// Mitsubishi GX Works2 project: BookEX6_13 Timer   PLC: Q13UDV

// global labels: Global
VAR_GLOBAL
  bVar0 AT M5000 : BOOL;
  abArray0 AT M5010 : ARRAY [0..49] OF BOOL;
  sStr0 AT D5000 : STRING[199];
  sStr1 AT D5100 : STRING[199];
  sStr2 AT D5200 : STRING[199];
  sStr3 AT D5300 : STRING[199];
  sStr4 AT D5400 : STRING[199];
  sStr5 AT D5500 : STRING[199];
  sStr6 AT D5600 : STRING[199];
  sStr7 AT D5700 : STRING[199];
  sStr8 AT D5800 : STRING[199];
  sStr9 AT D5900 : STRING[199];
  iVar0 AT D4500 : INT;
  iVar1 AT D4501 : INT;
  iVar2 AT D4502 : INT;
  iVar3 AT D4503 : INT;
  iVar4 AT D4504 : INT;
  iVar5 AT D4505 : INT;
  iVar6 AT D4506 : INT;
  iVar7 AT D4507 : INT;
  iVar8 AT D4508 : INT;
  iVar9 AT D4509 : INT;
  dVar0 AT D4510 : DINT;
  dVar1 AT D4512 : DINT;
  dVar2 AT D4514 : DINT;
  dVar3 AT D4516 : DINT;
  dVar4 AT D4518 : DINT;
  dVar5 AT D4520 : DINT;
  dVar6 AT D4522 : DINT;
  dVar7 AT D4524 : DINT;
  dVar8 AT D4526 : DINT;
  dVar9 AT D4528 : DINT;
  wVar0 AT D4530 : WORD;
  wVar1 AT D4531 : WORD;
  wVar2 AT D4532 : WORD;
  wVar3 AT D4533 : WORD;
  wVar4 AT D4534 : WORD;
  wVar5 AT D4535 : WORD;
  wVar6 AT D4536 : WORD;
  wVar7 AT D4537 : WORD;
  wVar8 AT D4538 : WORD;
  wVar9 AT D4539 : WORD;
  dwVar0 AT D4540 : DWORD;
  dwVar1 AT D4542 : DWORD;
  dwVar2 AT D4544 : DWORD;
  dwVar3 AT D4546 : DWORD;
  dwVar4 AT D4548 : DWORD;
  dwVar5 AT D4550 : DWORD;
  dwVar6 AT D4552 : DWORD;
  dwVar7 AT D4554 : DWORD;
  dwVar8 AT D4556 : DWORD;
  dwVar9 AT D4558 : DWORD;
  fsVar0 AT D4560 : REAL;
  fsVar1 AT D4562 : REAL;
  fsVar2 AT D4564 : REAL;
  fsVar3 AT D4566 : REAL;
  fsVar4 AT D4568 : REAL;
  fsVar5 AT D4570 : REAL;
  fsVar6 AT D4572 : REAL;
  fsVar7 AT D4574 : REAL;
  fsVar8 AT D4576 : REAL;
  fsVar9 AT D4578 : REAL;
  fdVar0 AT D4580 : LREAL;
  tTime0 AT D4620 : TIME;
  tTime1 AT D4622 : TIME;
  tTime2 AT D4624 : TIME;
  tTime3 AT D4626 : TIME;
  tTime4 AT D4628 : TIME;
  tTime5 AT D4630 : TIME;
  tTime6 AT D4632 : TIME;
  tTime7 AT D4634 : TIME;
  tTime8 AT D4636 : TIME;
  tTime9 AT D4638 : TIME;
  tTime10 AT D4640 : TIME;
  bVar1 AT M5001 : BOOL;
  bVar2 AT M5002 : BOOL;
  bVar3 AT M5003 : BOOL;
  bVar4 AT M5004 : BOOL;
  bVar5 AT M5005 : BOOL;
  bVar6 AT M5006 : BOOL;
  bVar7 AT M5007 : BOOL;
  bVar8 AT M5008 : BOOL;
  bVar9 AT M5009 : BOOL;
  abArray1 AT M5060 : ARRAY [0..49] OF BOOL;
  abArray2 AT M5110 : ARRAY [0..49] OF BOOL;
  abArray3 AT M5160 : ARRAY [0..49] OF BOOL;
  abArray4 AT M5210 : ARRAY [0..49] OF BOOL;
  abArray5 AT M5260 : ARRAY [0..49] OF BOOL;
  abArray6 AT M5310 : ARRAY [0..49] OF BOOL;
  abArray7 AT M5360 : ARRAY [0..49] OF BOOL;
  abArray8 AT M5410 : ARRAY [0..49] OF BOOL;
  abArray9 AT M5460 : ARRAY [0..49] OF BOOL;
  fdVar1 AT D4584 : LREAL;
  fdVar2 AT D4588 : LREAL;
  fdVar3 AT D4592 : LREAL;
  fdVar4 AT D4596 : LREAL;
  fdVar5 AT D4600 : LREAL;
  fdVar6 AT D4604 : LREAL;
  fdVar7 AT D4608 : LREAL;
  fdVar8 AT D4612 : LREAL;
  fdVar9 AT D4616 : LREAL;
  aSendData1 AT D100 : ARRAY [0..9] OF INT;
  aiTxData AT D4000 : ARRAY [0..99] OF INT;
  aiRxData AT D4100 : ARRAY [0..99] OF INT;
  iOpenOK AT D3900 : INT;
  iOpenERR AT D3901 : INT;
  iSendOK AT D3902 : INT;
  iSendERR AT D3903 : INT;
  iCloseOK AT D3906 : INT;
  iCloseERR AT D3907 : INT;
  iRecvOK AT D3904 : INT;
  iRecvERR AT D3905 : INT;
  aiTxData2 AT D4200 : ARRAY [0..99] OF INT;
  aiRxData2 AT D4300 : ARRAY [0..99] OF INT;
  iOpenOK2 AT D3908 : INT;
  iOpenERR2 AT D3909 : INT;
  iSendOK2 AT D3910 : INT;
  iSendERR2 AT D3911 : INT;
  iRecvOK2 AT D3912 : INT;
  iRecvERR2 AT D3913 : INT;
  iCloseOK2 AT D3914 : INT;
  iCloseERR2 AT D3915 : INT;
  iEOpenComp AT D3916 : INT;
  iEOpenReq AT D3917 : INT;
  iERecvFlag AT D3918 : INT;
  iOpenCode AT D3919 : INT;
  iSendCode AT D3920 : INT;
  iRecvCode AT D3921 : INT;
  iCloseCode AT D3922 : INT;
  iOpenCode2 AT D3923 : INT;
  iSendCode2 AT D3924 : INT;
  iRecvCode2 AT D3925 : INT;
  iCloseCode2 AT D3926 : INT;
  aRecvData1 AT D110 : ARRAY [0..9] OF INT;
  aSendData2 AT D120 : ARRAY [0..9] OF INT;
  aRecvData2 AT D130 : ARRAY [0..9] OF INT;
END_VAR
// user libraries (not included): HMI

FUNCTION_BLOCK BlinkFlag
VAR_INPUT
  b_EN : BOOL;
END_VAR
VAR_OUTPUT
  b_ENO : BOOL;
END_VAR
VAR
  bBlink : BOOL;
  fbTimer1 : TON;
  fbTimer2 : TON;
  BlinkTime : TIME;
END_VAR
VAR_OUTPUT
  t_ON : TIME;
  t_OFF : TIME;
END_VAR
VAR_INPUT
  i_Duty : INT;
END_VAR
VAR_OUTPUT
  b_Q : BOOL;
END_VAR
b_ENO := b_EN;
IF NOT b_EN THEN
	b_Q := FALSE;
	bBlink := FALSE;
	fbTimer1(IN:=FALSE);
	fbTimer2(IN:=FALSE);
	RETURN;
END_IF;
BlinkTime := INT_TO_TIME(i_Duty*100/2);
IF bBlink THEN
		fbTimer1(IN := TRUE , PT:=BlinkTime);
		IF fbTimer1.Q THEN
			bBlink := FALSE;
			fbTimer1(IN:=FALSE);
		END_IF;
ELSE
		fbTimer2(IN := TRUE , PT:=BlinkTime);
		IF fbTimer2.Q THEN
			bBlink := TRUE;
			fbTimer2(IN:=FALSE);
		END_IF;
END_IF;
b_Q := bBlink;
t_ON := fbTimer2.ET;
t_OFF := fbTimer1.ET;
END_FUNCTION_BLOCK

FUNCTION_BLOCK CntClick
VAR_INPUT
  b_IN : BOOL;
  i_IN : INT;
  t_Time : TIME;
END_VAR
VAR_OUTPUT
  b_Q : BOOL;
END_VAR
VAR
  oldIN : BOOL;
  iCnt : INT;
  fbTP : TP;
END_VAR
VAR_OUTPUT
  t_ET : TIME;
  i_Cnt : INT;
END_VAR
;
b_Q := FALSE;

IF b_IN AND NOT oldIN AND NOT fbTP.Q THEN
	iCnt := 1;
ELSIF fbTP.Q AND b_IN AND NOT oldIN THEN
	iCnt := iCnt + 1;
ELSIF NOT fbTP.Q THEN
	b_Q := iCnt = i_IN;
	iCnt := 0;
END_IF;

oldIN := b_IN;
fbTP(IN := b_IN, PT := t_Time);
t_ET := fbTP.ET;
i_Cnt := iCnt;
END_FUNCTION_BLOCK

FUNCTION_BLOCK DelayOut
VAR_INPUT
  b_SET : BOOL;
  b_RST : BOOL;
  b_IN : BOOL;
  t_Time : TIME;
END_VAR
VAR_OUTPUT
  b_Q : BOOL;
END_VAR
VAR
  fbTON : TON;
  bOld : BOOL;
END_VAR
;
IF fbTON.Q THEN b_Q := FALSE; END_IF;
IF b_RST THEN
	b_Q := FALSE;
ELSIF b_SET THEN
	b_Q := TRUE;
ELSIF b_IN AND NOT bOld THEN
	b_Q := TRUE; 
END_IF;
bOld := b_IN;
IF t_Time > T#0s THEN fbTON(IN := b_Q, PT := t_Time); END_IF;
END_FUNCTION_BLOCK

FUNCTION_BLOCK FlashLamp
VAR_INPUT
  t_OnTime : TIME;
  t_OffTime : TIME;
END_VAR
VAR_OUTPUT
  b_Lamp : BOOL;
END_VAR
VAR
  bFeed : BOOL;
  TON_1 : TON;
  TON_2 : TON;
END_VAR
VAR_OUTPUT
  t_Time0 : TIME;
  t_Time1 : TIME;
END_VAR
(* structured ladder/FBD written out as ST: instructions are called as NAME(EN, inputs, outputs); _pN, _eN, _tN stand for wires *)
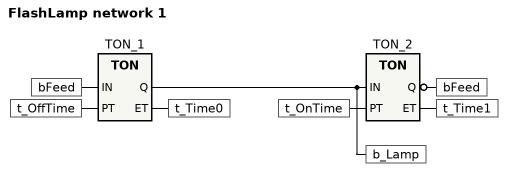
(* network 1 *)
TON_1(IN := bFeed, PT := t_OffTime, ET => t_Time0);
b_Lamp := TON_1.Q;
TON_2(IN := TON_1.Q, PT := t_OnTime, ET => t_Time1);
bFeed := NOT TON_2.Q;
END_FUNCTION_BLOCK

FUNCTION_BLOCK Flicker
VAR_INPUT
  t_Duty : TIME;
END_VAR
VAR_OUTPUT
  b_Lamp1 : BOOL;
  b_Lamp2 : BOOL;
END_VAR
VAR
  bRes : BOOL;
  iInterval : INT;
  tTimer0 : TIMER;
  tTimer1 : TIMER;
END_VAR
;
iInterval := TIME_TO_INT(t_Duty) / 100;
bResult := OUT_T(NOT tTimer1.S, tTimer0, iInterval);
bResult := OUT_T(tTimer0.S, tTimer1, iInterval);
b_Lamp1 := tTimer0.S;
b_Lamp2 :=   NOT tTimer0.S;
END_FUNCTION_BLOCK

FUNCTION_BLOCK HeartBeat
VAR_INPUT
  t_TxTime : TIME;
END_VAR
VAR_OUTPUT
  b_ENO : BOOL;
  b_TxFlag : BOOL;
END_VAR
VAR
  SeqTx : INT;
  fbTxTimer : TON;
END_VAR
VAR_INPUT
  t_RxTime : TIME;
  b_RxFlag : BOOL;
END_VAR
VAR_OUTPUT
  b_RxError : BOOL;
END_VAR
VAR
  fbRxTimer : TON;
  oldRxFlag : BOOL;
END_VAR
VAR_INPUT
  b_EN : BOOL;
END_VAR
VAR_OUTPUT
  b_TxChanged : BOOL;
END_VAR
;
b_ENO := b_EN;
IF NOT b_EN THEN
	SeqTx := 0;
	b_TxFlag := FALSE;
	b_RxError := FALSE;
	RETURN;
END_IF;
	
CASE SeqTx OF
			0 : 
				b_TxFlag := TRUE;
				SeqTx := 1;
				b_TxChanged := TRUE;
			1 : 
				b_TxChanged := FALSE;
				fbTxTimer(IN := TRUE , PT := t_TxTime);
				IF fbTxTimer.Q THEN
					fbTxTimer(IN := FALSE);
					SeqTx := 2;
				END_IF;
			2 : 
				b_TxFlag := FALSE;
				SeqTx := 3;
				b_TxChanged := TRUE;
			3 : 
				b_TxChanged := FALSE;
				fbTxTimer(IN := TRUE , PT := t_TxTime);
				IF fbTxTimer.Q THEN
					fbTxTimer(IN := FALSE);
					SeqTx := 0;
				END_IF;
ELSE
			    SeqTx := 0;
END_CASE;

IF b_RxFlag = oldRxFlag THEN
			fbRxTimer(IN := TRUE ,  PT := t_RxTime);
			IF fbRxTimer.Q THEN
				fbRxTimer(IN := FALSE);
				b_RxError := TRUE;
			END_IF;
ELSE
			fbRxTimer(IN := FALSE);
			oldRxFlag := b_RxFlag;
			b_RxError := FALSE;
END_IF;
END_FUNCTION_BLOCK

FUNCTION_BLOCK Interlock
VAR_INPUT
  b_IN1 : BOOL;
  b_IN2 : BOOL;
  t_Time : TIME;
END_VAR
VAR_OUTPUT
  b_Q1 : BOOL;
  b_Q2 : BOOL;
END_VAR
VAR
  fbTOF1 : TOF;
  fbTOF2 : TOF;
END_VAR
VAR_OUTPUT
  t_ET1 : TIME;
  t_ET2 : TIME;
END_VAR
;
fbTOF1(IN := b_IN1, PT := t_Time);
fbTOF2(IN := b_IN2, PT := t_Time);

b_Q1 := b_IN1 AND NOT fbTOF2.Q;
b_Q2 := b_IN2 AND NOT fbTOF1.Q;
t_ET1 := fbTOF1.ET;
t_ET2 := fbTOF2.ET;
END_FUNCTION_BLOCK

FUNCTION_BLOCK TONOF
VAR_INPUT
  b_IN : BOOL;
  t_ON : TIME;
  t_OFF : TIME;
END_VAR
VAR_OUTPUT
  b_Q : BOOL;
END_VAR
VAR
  fbTON : TON;
  bOld : BOOL;
  bMode : BOOL;
END_VAR
VAR_OUTPUT
  t_ET : TIME;
END_VAR
;
IF b_IN XOR bOld THEN
  fbTON(IN := FALSE, PT := SEL(b_IN, t_OFF, t_ON));
  bMode := b_IN;
  bOld := b_IN;
END_IF;
fbTON(IN := TRUE);
IF fbTON.Q THEN 
	b_Q := bMode;
END_IF;
t_ET := fbTON.ET;
END_FUNCTION_BLOCK

PROGRAM ExBlink
VAR
  HMI03_1 : HMI03;
  BlinkFlag_2 : BlinkFlag;
END_VAR
(* structured ladder/FBD written out as ST: instructions are called as NAME(EN, inputs, outputs); _pN, _eN, _tN stand for wires *)
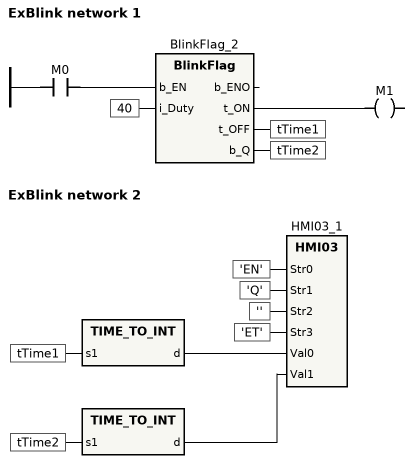
(* network 1 *)
BlinkFlag_2(b_EN := M0, i_Duty := 40, t_OFF => tTime1, b_Q => tTime2);
M1 := BlinkFlag_2.t_ON;
(* network 2 *)
HMI03_1(Str0 := 'EN', Str1 := 'Q', Str2 := '', Str3 := 'ET', Val0 := TIME_TO_INT(tTime1), Val1 := TIME_TO_INT(tTime2));
END_PROGRAM

PROGRAM ExCntClick
VAR
  CntClick_1 : CntClick;
  TP_1 : TP;
  HMI03_1 : HMI03;
END_VAR
(* structured ladder/FBD written out as ST: instructions are called as NAME(EN, inputs, outputs); _pN, _eN, _tN stand for wires *)
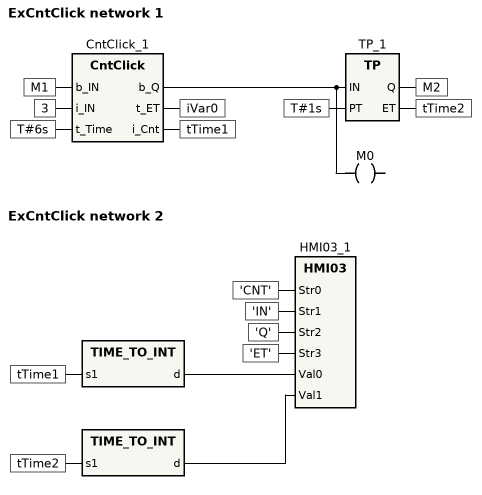
(* network 1 *)
CntClick_1(b_IN := M1, i_IN := 3, t_Time := T#6s, t_ET => iVar0, i_Cnt => tTime1);
M0 := CntClick_1.b_Q;
TP_1(IN := CntClick_1.b_Q, PT := T#1s, Q => M2, ET => tTime2);
(* network 2 *)
HMI03_1(Str0 := 'CNT', Str1 := 'IN', Str2 := 'Q', Str3 := 'ET', Val0 := TIME_TO_INT(tTime1), Val1 := TIME_TO_INT(tTime2));
END_PROGRAM

PROGRAM ExDelayOut
VAR
  DelayOut_1 : DelayOut;
  HMI05_1 : HMI05;
END_VAR
(* structured ladder/FBD written out as ST: instructions are called as NAME(EN, inputs, outputs); _pN, _eN, _tN stand for wires *)
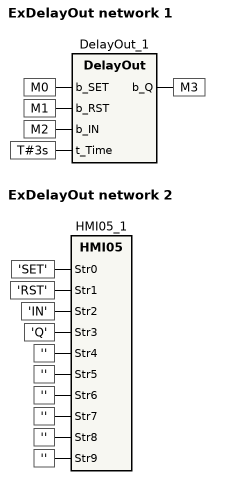
(* network 1 *)
DelayOut_1(b_SET := M0, b_RST := M1, b_IN := M2, t_Time := T#3s, b_Q => M3);
(* network 2 *)
HMI05_1(Str0 := 'SET', Str1 := 'RST', Str2 := 'IN', Str3 := 'Q', Str4 := '', Str5 := '', Str6 := '', Str7 := '', Str8 := '', Str9 := '');
END_PROGRAM

PROGRAM ExFlash
VAR
  FlashLamp_1 : FlashLamp;
  HMI03_1 : HMI03;
END_VAR
(* structured ladder/FBD written out as ST: instructions are called as NAME(EN, inputs, outputs); _pN, _eN, _tN stand for wires *)
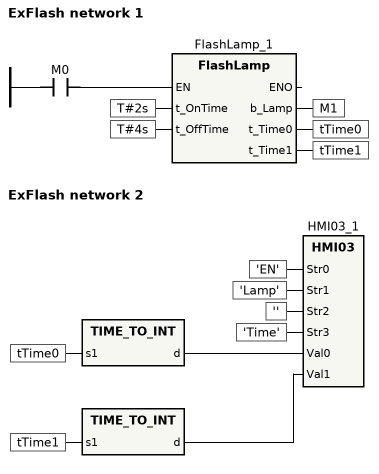
(* network 1 *)
FlashLamp_1(EN := M0, t_OnTime := T#2s, t_OffTime := T#4s, b_Lamp => M1, t_Time0 => tTime0, t_Time1 => tTime1);
(* network 2 *)
HMI03_1(Str0 := 'EN', Str1 := 'Lamp', Str2 := '', Str3 := 'Time', Val0 := TIME_TO_INT(tTime0), Val1 := TIME_TO_INT(tTime1));
END_PROGRAM

PROGRAM ExHeartBeat
VAR
  HeartBeat_1 : HeartBeat;
  HMI05_1 : HMI05;
  k_FWD : BOOL;
  k_BWD : BOOL;
  o_FWD : BOOL;
  o_BWD : BOOL;
END_VAR
(* structured ladder/FBD written out as ST: instructions are called as NAME(EN, inputs, outputs); _pN, _eN, _tN stand for wires *)
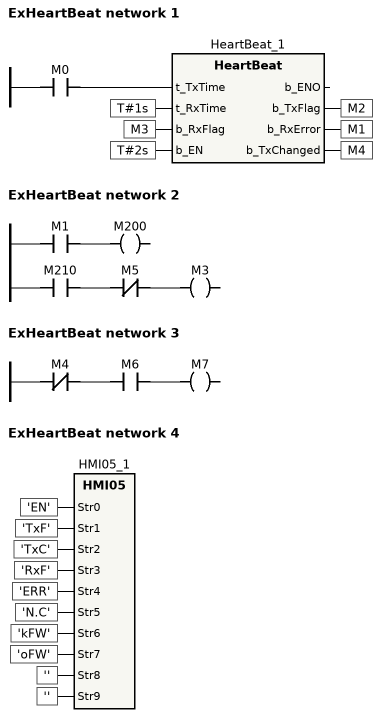
(* network 1 *)
HeartBeat_1(t_TxTime := M0, t_RxTime := T#1s, b_RxFlag := M3, b_EN := T#2s, b_TxFlag => M2, b_RxError => M1, b_TxChanged => M4);
(* network 2 *)
M200 := M1;
M3 := M210 AND NOT M5;
(* network 3 *)
M7 := NOT M4 AND M6;
(* network 4 *)
HMI05_1(Str0 := 'EN', Str1 := 'TxF', Str2 := 'TxC', Str3 := 'RxF', Str4 := 'ERR', Str5 := 'N.C', Str6 := 'kFW', Str7 := 'oFW', Str8 := '', Str9 := '');
END_PROGRAM

PROGRAM ExInterlock
VAR
  Interlock_1 : Interlock;
  HMI02_1 : HMI02;
END_VAR
(* structured ladder/FBD written out as ST: instructions are called as NAME(EN, inputs, outputs); _pN, _eN, _tN stand for wires *)
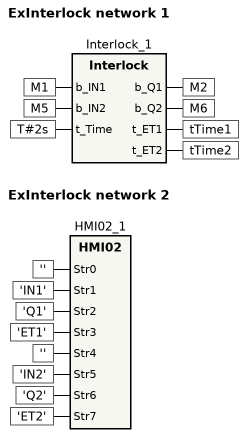
(* network 1 *)
Interlock_1(b_IN1 := M1, b_IN2 := M5, t_Time := T#2s, b_Q1 => M2, b_Q2 => M6, t_ET1 => tTime1, t_ET2 => tTime2);
(* network 2 *)
HMI02_1(Str0 := '', Str1 := 'IN1', Str2 := 'Q1', Str3 := 'ET1', Str4 := '', Str5 := 'IN2', Str6 := 'Q2', Str7 := 'ET2');
END_PROGRAM

PROGRAM ExTIMER
VAR
  TIMER_10_FB_M_1 : TIMER_10_FB_M;
  TIMER_LOW_FB_M_1 : TIMER_LOW_FB_M;
  TIMER_CONT_FB_M_1 : TIMER_CONT_FB_M;
  TIMER_100_FB_M_1 : TIMER_100_FB_M;
  TIMER_HIGH_FB_M_1 : TIMER_HIGH_FB_M;
  TIMER_CONT_FB_M_2 : TIMER_CONT_FB_M;
  TIMER_CONTHFB_M_1 : TIMER_CONTHFB_M;
END_VAR
(* structured ladder/FBD written out as ST: instructions are called as NAME(EN, inputs, outputs); _pN, _eN, _tN stand for wires *)
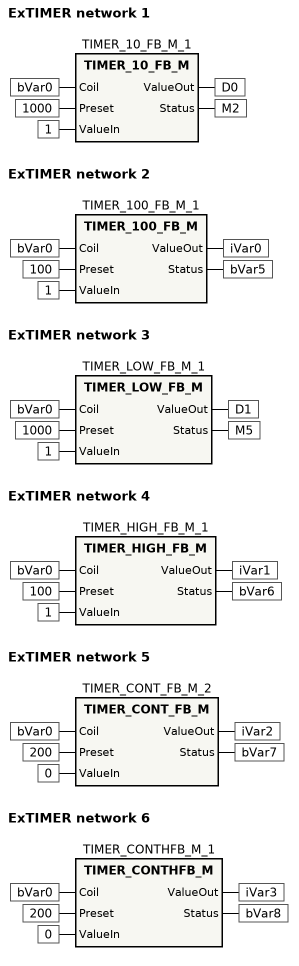
(* network 1 *)
TIMER_10_FB_M_1(Coil := bVar0, Preset := 1000, ValueIn := 1, ValueOut => D0, Status => M2);
(* network 2 *)
TIMER_100_FB_M_1(Coil := bVar0, Preset := 100, ValueIn := 1, ValueOut => iVar0, Status => bVar5);
(* network 3 *)
TIMER_LOW_FB_M_1(Coil := bVar0, Preset := 1000, ValueIn := 1, ValueOut => D1, Status => M5);
(* network 4 *)
TIMER_HIGH_FB_M_1(Coil := bVar0, Preset := 100, ValueIn := 1, ValueOut => iVar1, Status => bVar6);
(* network 5 *)
TIMER_CONT_FB_M_2(Coil := bVar0, Preset := 200, ValueIn := 0, ValueOut => iVar2, Status => bVar7);
(* network 6 *)
TIMER_CONTHFB_M_1(Coil := bVar0, Preset := 200, ValueIn := 0, ValueOut => iVar3, Status => bVar8);
END_PROGRAM

PROGRAM ExTOF
VAR
  TOF_E_1 : TOF_E;
  HMI03_1 : HMI03;
END_VAR
(* structured ladder/FBD written out as ST: instructions are called as NAME(EN, inputs, outputs); _pN, _eN, _tN stand for wires *)
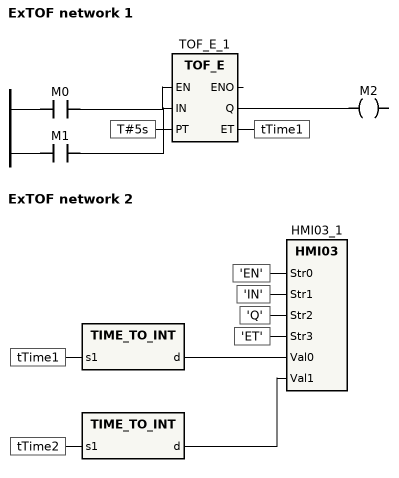
(* network 1 *)
TOF_E_1(EN := M0, IN := M1, PT := T#5s, ET => tTime1);
M2 := TOF_E_1.Q;
(* network 2 *)
HMI03_1(Str0 := 'EN', Str1 := 'IN', Str2 := 'Q', Str3 := 'ET', Val0 := TIME_TO_INT(tTime1), Val1 := TIME_TO_INT(tTime2));
END_PROGRAM

PROGRAM ExTON
VAR
  TON_E_1 : TON_E;
  HMI03_1 : HMI03;
END_VAR
(* structured ladder/FBD written out as ST: instructions are called as NAME(EN, inputs, outputs); _pN, _eN, _tN stand for wires *)
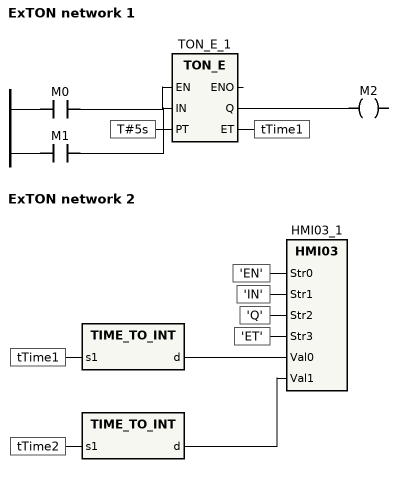
(* network 1 *)
TON_E_1(EN := M0, IN := M1, PT := T#5s, ET => tTime1);
M2 := TON_E_1.Q;
(* network 2 *)
HMI03_1(Str0 := 'EN', Str1 := 'IN', Str2 := 'Q', Str3 := 'ET', Val0 := TIME_TO_INT(tTime1), Val1 := TIME_TO_INT(tTime2));
END_PROGRAM

PROGRAM ExTON2
VAR
  TON_1 : TON;
  TON_2 : TON;
  HMI02_1 : HMI02;
END_VAR
(* structured ladder/FBD written out as ST: instructions are called as NAME(EN, inputs, outputs); _pN, _eN, _tN stand for wires *)
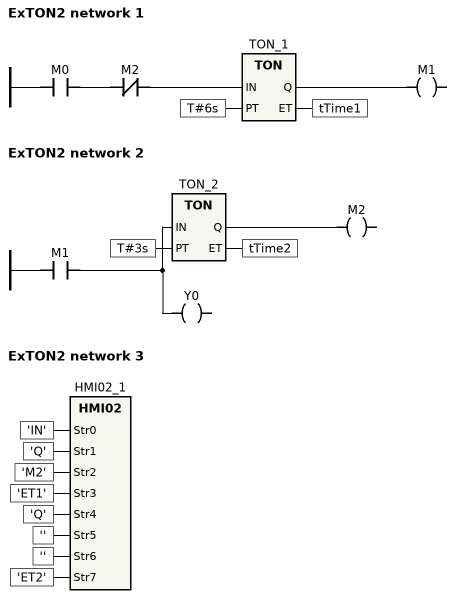
(* network 1 *)
TON_1(IN := M0 AND NOT M2, PT := T#6s, ET => tTime1);
M1 := TON_1.Q;
(* network 2 *)
TON_2(IN := M1, PT := T#3s, ET => tTime2);
M2 := TON_2.Q;
Y0 := M1;
(* network 3 *)
HMI02_1(Str0 := 'IN', Str1 := 'Q', Str2 := 'M2', Str3 := 'ET1', Str4 := 'Q', Str5 := '', Str6 := '', Str7 := 'ET2');
END_PROGRAM

PROGRAM ExTON3
VAR
  TON_1 : TON;
  TON_2 : TON;
  HMI02_1 : HMI02;
END_VAR
(* structured ladder/FBD written out as ST: instructions are called as NAME(EN, inputs, outputs); _pN, _eN, _tN stand for wires *)
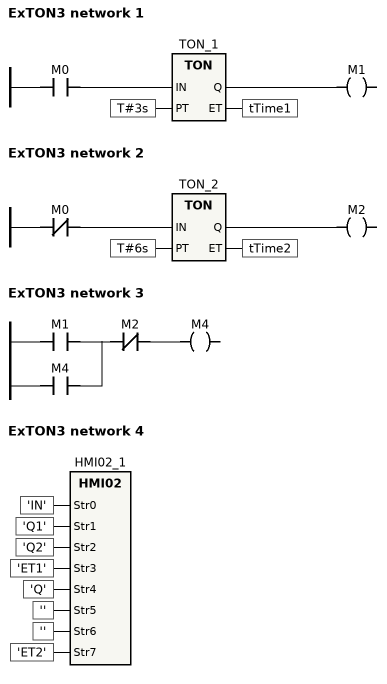
(* network 1 *)
TON_1(IN := M0, PT := T#3s, ET => tTime1);
M1 := TON_1.Q;
(* network 2 *)
TON_2(IN := NOT M0, PT := T#6s, ET => tTime2);
M2 := TON_2.Q;
(* network 3 *)
M4 := (M1 OR M4) AND NOT M2;
(* network 4 *)
HMI02_1(Str0 := 'IN', Str1 := 'Q1', Str2 := 'Q2', Str3 := 'ET1', Str4 := 'Q', Str5 := '', Str6 := '', Str7 := 'ET2');
END_PROGRAM

PROGRAM ExTON4
VAR
  TON_1 : TON;
  TON_2 : TON;
  HMI02_1 : HMI02;
END_VAR
(* structured ladder/FBD written out as ST: instructions are called as NAME(EN, inputs, outputs); _pN, _eN, _tN stand for wires *)
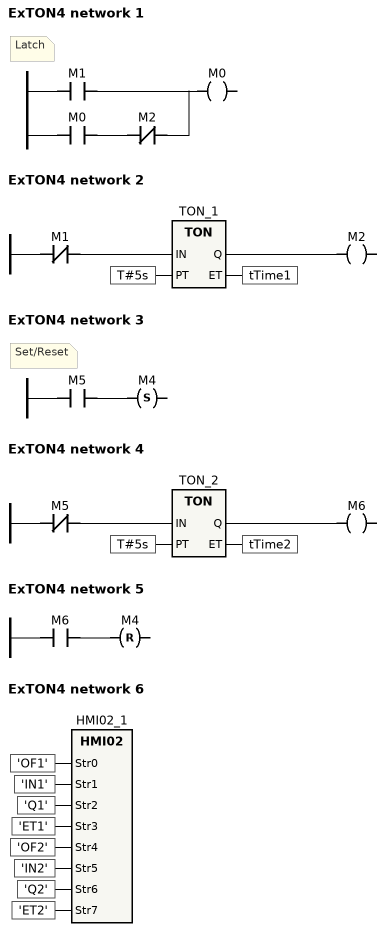
(* network 1 *)
(* Latch *)
M0 := M1 OR (M0 AND NOT M2);
(* network 2 *)
TON_1(IN := NOT M1, PT := T#5s, ET => tTime1);
M2 := TON_1.Q;
(* network 3 *)
(* Set/Reset *)
SET(M5, M4);
(* network 4 *)
TON_2(IN := NOT M5, PT := T#5s, ET => tTime2);
M6 := TON_2.Q;
(* network 5 *)
RST(M6, M4);
(* network 6 *)
HMI02_1(Str0 := 'OF1', Str1 := 'IN1', Str2 := 'Q1', Str3 := 'ET1', Str4 := 'OF2', Str5 := 'IN2', Str6 := 'Q2', Str7 := 'ET2');
END_PROGRAM

PROGRAM ExTONOF
VAR
  TONOF_1 : TONOF;
  HMI03_1 : HMI03;
END_VAR
(* structured ladder/FBD written out as ST: instructions are called as NAME(EN, inputs, outputs); _pN, _eN, _tN stand for wires *)
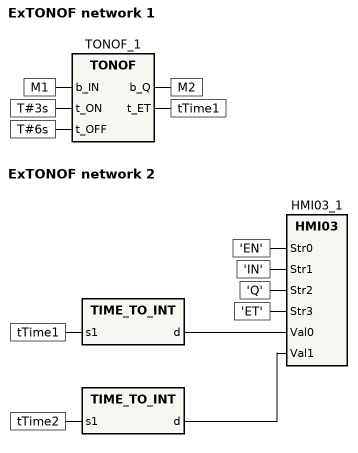
(* network 1 *)
TONOF_1(b_IN := M1, t_ON := T#3s, t_OFF := T#6s, b_Q => M2, t_ET => tTime1);
(* network 2 *)
HMI03_1(Str0 := 'EN', Str1 := 'IN', Str2 := 'Q', Str3 := 'ET', Val0 := TIME_TO_INT(tTime1), Val1 := TIME_TO_INT(tTime2));
END_PROGRAM

PROGRAM ExTP
VAR
  TP_E_1 : TP_E;
  TP_1 : TP;
  HMI03_1 : HMI03;
END_VAR
(* structured ladder/FBD written out as ST: instructions are called as NAME(EN, inputs, outputs); _pN, _eN, _tN stand for wires *)
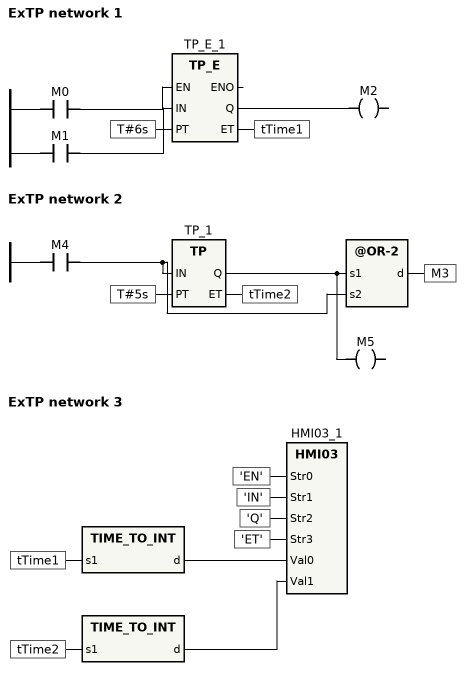
(* network 1 *)
TP_E_1(EN := M0, IN := M1, PT := T#6s, ET => tTime1);
M2 := TP_E_1.Q;
(* network 2 *)
TP_1(IN := M4, PT := T#5s, ET => tTime2);
M5 := TP_1.Q;
M3 := @OR-2(TP_1.Q, M4);
(* network 3 *)
HMI03_1(Str0 := 'EN', Str1 := 'IN', Str2 := 'Q', Str3 := 'ET', Val0 := TIME_TO_INT(tTime1), Val1 := TIME_TO_INT(tTime2));
END_PROGRAM

FUNCTION_BLOCK Bounce
VAR_INPUT
  IN : BOOL;
  PT_On : TIME;
  PT_Off : TIME;
END_VAR
VAR_OUTPUT
  iOUT : BOOL;
END_VAR
VAR
  fbOnTimer : TON;
  fbOffTimer : TOF;
  dOn : TIME;
  dOff : TIME;
END_VAR
;
(*
IF PT_ON < T#500ms THEN
	dOn := T#500ms;
ELSE
	dOn := PT_ON;
END_IF;

IF PT_OFF < T#500ms THEN
	dOff := T#500ms;
ELSE
	dOff := PT_OFF;
END_IF;
*)
dOn := PT_On;
dOff := PT_Off;
fbOnTimer(IN := IN , PT := dOn);
fbOffTimer(IN := fbOnTimer.Q , PT := dOff);
iOUT := fbOffTimer.Q;
tTime1 := fbOnTimer.ET;
tTime2 := fbOffTimer.ET;
END_FUNCTION_BLOCK

PROGRAM ExTitle
VAR
  TON_1 : TON;
  TON_2 : TON;
END_VAR
(* structured ladder/FBD written out as ST: instructions are called as NAME(EN, inputs, outputs); _pN, _eN, _tN stand for wires *)
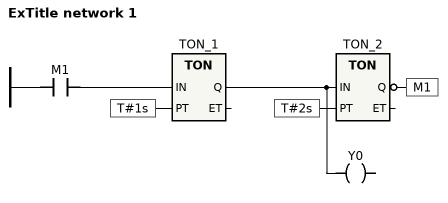
(* network 1 *)
TON_1(IN := M1, PT := T#1s);
Y0 := TON_1.Q;
TON_2(IN := TON_1.Q, PT := T#2s);
M1 := NOT TON_2.Q;
END_PROGRAM
